FUNCTION_BLOCK FB_Gantry
VAR CONSTANT
	sCycleStateTextDef: ARRAY[0..10]  OF STRING :=	
		['State 0: Wait for Start','1','2','3','4','5','6','7','8','9',
		'State 10: Error'];
	
	tCycleStateTimeouts: ARRAY[0..10] OF TIME := 
		[T#10S,T#10S,T#10S,T#10S,T#10S,T#10S,T#10S,T#10S,T#10S,T#10S,
		T#10S];

	sInitStateTextDef: ARRAY[0..10] OF STRING :=
		['State 0: Wait for Start',
		'State 1: Description Init State 1',
		'State 2: Description Init State 2',
		'State 3; Description Init State 3',
		'State 4; Description Init State 4',
		'State 5; Description Init State 5',
		'State 6; Error State'];

	tInitStateTimeouts: ARRAY[0..10] OF TIME := 
		[T#10S,T#10S,T#10S,T#10S,T#10S,T#10S,T#10S,T#10S,T#10S,T#10S
		,T#10S];
END_VAR
VAR_INPUT
	mxResetCycleState				: BOOL;
	mxResetInitState				: BOOL;
	mxForceInit						: BOOL; (*Reset Calibration Flag*)
	mxReset							: BOOL;	(*Reset Error*)
	mxEmergency						: BOOL;
	mxAutoMode						: BOOL; (* TRUE = Automode *)
	mxFirstCycle					: BOOL;

	mrModPosConveyor				: LREAL;
	mxProductReadyAtTakeout			: BOOL; (* Signal from BottomMold, Takeout Unit *)
	mxDisableCollision				: BOOL;
END_VAR
VAR_IN_OUT
	MachParameters					: ST_GantryMachPar;
	ProdParameters					: ST_GantryProdPar;
	SysParameters					: ST_GantrySysPar;
END_VAR
VAR_OUTPUT
	(*Errors*)
	Errors							: ST_GantryErrors;
	mxErrorInit						: BOOL;		(* Error, stop immediately. Initialisation neccesary *)
	mxErrorStopinPos				: BOOL;		(* Error, stop in position. Only reset neccesary *)

(* State vars *)
	mxCycleBusy						: BOOL;
	mxInitBusy						: BOOL;
	
(* Vars *)
	mxInitialized					: BOOL;
	mrActPosHorizontal				: LREAL;
	mrActPosVertical				: LREAL;
	mxHorizontalIsMoving			: BOOL;
	mxVerticalIsMoving				: BOOL;
	
	(* Signals *)
	mxIsEmpty						: BOOL;
	mxProductPickedUp				: BOOL;
END_VAR
VAR
(* State vars *)
	miCycleState					: INT :=0;
	miCycleOldstate					: INT :=0;
	mxCycleTransitionState			: BOOL := FALSE;
	sCycleStateText					: STRING;
	exCycleTimeOut					: BOOL;		(* Timeout for the whole programcycle *)
	CycleTimeout					: TON;
	CycleTimeOutUpFlank				: R_TRIG;
	mxCycleTimeoutEnable			: BOOL;
	CycleTime						: REAL;
	mxCycleHasError					: BOOL;
	miStopState						: INT;
	mxStartCycle					: BOOL;
	mxStopCycle						: BOOL;
	mxStopDirect					: BOOL;
	
	miInitState						: INT	:=0;
	miInitOldstate					: INT	:=0;
	mxInitTransitionState			: BOOL	:= FALSE;
	sInitStateText					: STRING;
	exInitTimeOut					: BOOL;		(* Timeout for the whole programcycle *)
	InitTimeout						: TON;
	InitTimeOutUpFlank				: R_TRIG;
	mxInitTimeoutEnable				: BOOL;
	InitTime						: REAL;
	mxInitHasError					: BOOL;
	mxStartInit						: BOOL;
	mxStopInit						: BOOL;

	ixCollision						AT %I*: BOOL;	(* Vertical axis *)
	ixEndLimitHorFront				AT %I*: BOOL;
	ixEndLimitHorBack				AT %I*: BOOL;
	ixEndLimitVertUp				AT %I*: BOOL;
	ixEndLimitVertDown				AT %I*: BOOL;
	
	(* Objects *)
	HorizontalAxis					: FB_NcAxis;
	VerticalAxis					: FB_NcAxis;
	(* Pickup Head *)
	BlowOff							: ARRAY [1..6] OF FB_MonoValveNoFdbck;
	VacuumValve						: ARRAY [1..6] OF FB_MonoValveNoFdbck;
	ixVacuumSensor					 AT %I* : ARRAY [1..6] OF BOOL;

(* Vars *)	
	miVacSection					: INT;
	miBlowOffSection				: INT;
	
	mxSwitchVacuumOn				: BOOL;
	(* Errors *)
	SR_exCollision					: SR;
	SR_exEndLimitHorFront			: SR;
	SR_exEndLimitHorBack			: SR;
	SR_exEndLimitVertUp				: SR;
	SR_exEndLimitVertDown			: SR;
	SR_exProductLost				: ARRAY [1..6] OF SR;
	T_VacSensor						: ARRAY [1..6] OF TON;
	mxSwitchBlowOffOn				: BOOL;
	T_WaitAtPickupPosition: TON;
	RT_DropOffPosCoveyor: R_TRIG;
	T_BlowOff: TON;
	mxTemp: BOOL;
	mxTemp2: BOOL;
	mxTest: BOOL;
	FT_SwitchVacuumOff: F_TRIG;
	FT_SwitchBlowOff: F_TRIG;
END_VAR

Error();
Cycle();
Init();
Objects();

ACTION Cycle:
(*StateChange (Transition)  Signalgeneration*)
mxCycleTransitionState:=(miCycleState<>miCycleOldstate);
(*State text*)
sCycleStateText:=sCycleStateTextDef[miCycleState];
(*Timeout Watchdog for Statemachine*)
mxCycleTimeoutEnable:=NOT (miCycleState=0) AND NOT mxReset;

CycleTimeout(IN:=mxCycleTimeoutEnable, PT:=tCycleStateTimeouts[miCycleState] );
CycleTimeOutUpFlank(CLK:=CycleTimeout.Q );
miCycleOldstate:=miCycleState;

(*Set Errorbit when Raising edge of Timeout has been detected*)
IF CycleTimeOutUpFlank.Q THEN
	exCycleTimeOut:=TRUE; 			(* 1 Timeout for the whole programcycle *)
END_IF

(*Function to reset the Statemachine*)
IF mxResetCycleState THEN
	mxResetCycleState:= FALSE;
	miCycleState:=0;
	miCycleOldstate:=miCycleState;
	mxCycleTransitionState:=FALSE;

	mxInitialized:= FALSE;
	mxStartCycle:= FALSE;
	mxStopCycle:= FALSE;
	mxStopDirect:= FALSE;

	mxIsEmpty:= FALSE;
	mxProductPickedUp:= FALSE;
	mxSwitchBlowOffOn:= FALSE;
	mxSwitchVacuumOn:= FALSE;

	T_WaitAtPickupPosition.IN:= FALSE;
	T_BlowOff.IN:= FALSE;
END_IF

fT_SwitchVacuumOff(CLK:= mxSwitchVacuumOn);
FT_SwitchBlowOff(CLK:=mxSwitchBlowOffOn);


(*Definition State has Error*)
mxCycleHasError:=FALSE;

// Open active valves on switch vacuum on.
IF (mxSwitchVacuumOn AND mxAutoMode) THEN
	IF MachParameters.EnableVacuumSection[1] THEN VacuumValve[1].M_On(); END_IF
	IF MachParameters.EnableVacuumSection[2] THEN VacuumValve[2].M_On(); END_IF
	IF MachParameters.EnableVacuumSection[3] THEN VacuumValve[3].M_On(); END_IF
	IF MachParameters.EnableVacuumSection[4] THEN VacuumValve[4].M_On(); END_IF
END_IF

// On trigger, close active valves
IF fT_SwitchVacuumOff.q AND mxAutoMode THEN
	IF MachParameters.EnableVacuumSection[1] THEN VacuumValve[1].M_Off(); END_IF
	IF MachParameters.EnableVacuumSection[2] THEN VacuumValve[2].M_Off(); END_IF
	IF MachParameters.EnableVacuumSection[3] THEN VacuumValve[3].M_Off(); END_IF
	IF MachParameters.EnableVacuumSection[4] THEN VacuumValve[4].M_Off(); END_IF
END_IF

// Open blowoff valves
IF mxSwitchBlowOffOn AND mxAutoMode THEN
	BlowOff[1].M_On();
	BlowOff[2].M_On();
	BlowOff[3].M_On();
	BlowOff[4].M_On();
END_IF

// On trigger, close blowoff valves.
IF FT_SwitchBlowOff.q AND mxAutoMode THEN
	BlowOff[1].M_Off();
	BlowOff[2].M_Off();
	BlowOff[3].M_Off();
	BlowOff[4].M_Off();
END_IF

RT_DropOffPosCoveyor(CLK:= mrModPosConveyor > MachParameters.DropOffConveyorPostion);
T_WaitAtPickupPosition(IN:= , PT:= T#1S);		
T_BlowOff(IN:= , PT:= ProdParameters.BlowOffTime);
IF T_BlowOff.Q THEN T_BlowOff.IN:= FALSE; END_IF
	
(*Cycle State's*)
CASE miCycleState OF
	0:
	(*
	
	- StopCyle en mxPause -> stop bewegingen.
	- Stop Cycle -> empty machine, ga naar rust
	
		- wait for startcycle
		- wait for product ready at takeout
		- Move horizontal to product pickup
		- move vertical to product pickup
		- Vacuum on
		- Move vertical up to transport pos
		- Move horizontal to drop off position (Rest)
		- wait for drop off position conveyor
		- Move vertical down to dropoff position
		- Blow off product
		- Move vertical up to transport pos
		- Goto 1

		* During vertical down, guard the collission sensor=> stop hor and vertical
		* Vacuum sensor check when vacuum on=> error leakage
		*  
	*)
		IF mxStartCycle THEN
			mxStartCycle:= FALSE;
			mxIsEmpty:= FALSE;
			mxProductPickedUp:= FALSE;

			miCycleState:= 1;
		END_IF	

	(* Set when goto 1 mxIsEmpty:= FALSE;	*)

	(* Wait for product ready at takeout *)
	1:
		IF mxStopDirect THEN
			mxStopDirect:= FALSE;
			
			miCycleState:= 25;
		//ELSIF mxStopCycle AND mxPause THEN
		//	mxPause:= FALSE;
			
		//	miCycleState:= 0;
		ELSIF mxStopCycle THEN
			mxStopCycle:= FALSE;
			VerticalAxis.M_Stop();
			HorizontalAxis.M_Stop();
			
			miStopState:= miCycleState;
			miCycleState:= 20;
		ELSIF mxProductReadyAtTakeout THEN
			mxProductReadyAtTakeout:= FALSE;
			mxIsEmpty:= FALSE;
			mxProductPickedUp:= FALSE;
			
			miCycleState:= 2;
		END_IF
		
	(* Move horizontal to the front to pickup position *)
	2:
		IF mxStopDirect THEN
			mxStopDirect:= FALSE;
			
			miCycleState:= 25;
		ELSIF mxStopCycle THEN
			mxStopCycle:= FALSE;
			VerticalAxis.M_Stop();
			HorizontalAxis.M_Stop();
			
			miStopState:= miCycleState;
			miCycleState:= 20;
		ELSIF HorizontalAxis.M_MoveAbsolute(Position:= MachParameters.PositionHorizontalPickup, Velocity:= MachParameters.Hor_VelocityAuto) THEN

			mxSwitchVacuumOn:= TRUE;
			
			miCycleState:=3;
		END_IF

	(* Move Vertical down to pickup position, vacuum on *)
	3:
		IF mxStopDirect THEN
			mxStopDirect:= FALSE;
			
			miCycleState:= 25;
		ELSIF mxStopCycle THEN
			mxStopCycle:= FALSE;
			
			miStopState:= miCycleState;
			miCycleState:= 20;
		ELSIF VerticalAxis.M_MoveAbsolute(Position:= ProdParameters.PositionVerticalPickup, Velocity:= MachParameters.Vert_VelocityAuto) THEN
		
			miCycleState:= 4;
		END_IF

	(* Wait at pickup position *)	
	4:
		T_WaitAtPickupPosition.IN:= TRUE;
	
		IF mxStopDirect THEN
			mxStopDirect:= FALSE;
			
			miCycleState:= 25;
		ELSIF mxStopCycle THEN
			mxStopCycle:= FALSE;
			
			miStopState:= miCycleState;
			miCycleState:= 20;
		ELSIF T_WaitAtPickupPosition.Q THEN
			T_WaitAtPickupPosition.IN:= FALSE;
			
			miCycleState:= 5;
		END_IF		

	(* Move Vertical up to transport position *)
	5:
		IF mxStopDirect THEN
			mxStopDirect:= FALSE;
			
			miCycleState:= 25;
		ELSIF mxStopCycle THEN
			mxStopCycle:= FALSE;
			
			miStopState:= miCycleState;
			miCycleState:= 20;
		ELSIF VerticalAxis.M_MoveAbsolute(Position:= MachParameters.Vert_PositionTransport, Velocity:= MachParameters.Vert_VelocityAuto) THEN
			mxProductPickedUp:= TRUE;

			miCycleState:= 6;
		END_IF
		
	(* Move horizontal to the back to drop-off position *)
	6:
		IF mxStopDirect THEN
			mxStopDirect:= FALSE;
			
			miCycleState:= 25;
		ELSIF mxStopCycle THEN
			mxStopCycle:= FALSE;
			
			miStopState:= miCycleState;
			miCycleState:= 20;
		ELSIF HorizontalAxis.M_MoveAbsolute(Position:= MachParameters.PositionHorizontalDropOff, Velocity:= MachParameters.Hor_VelocityAuto) THEN
			mxProductPickedUp := FALSE;
			miCycleState:= 7;
		END_IF
		
	(* Wait for drop off position conveyor *)
	7:
		IF mxStopDirect THEN
			mxStopDirect:= FALSE;
			
			miCycleState:= 25;
		ELSIF mxStopCycle THEN
			mxStopCycle:= FALSE;
			
			miStopState:= miCycleState;
			miCycleState:= 20;
		ELSIF RT_DropOffPosCoveyor.Q THEN
			
			miCycleState:= 8;
		END_IF

	(* Move Vertical Axis down to drop off position *)
	8:
		IF mxStopDirect THEN
			mxStopDirect:= FALSE;
			
			miCycleState:= 25;
		ELSIF mxStopCycle THEN
			mxStopCycle:= FALSE;
			
			miStopState:= miCycleState;
			miCycleState:= 20;
		ELSIF VerticalAxis.M_MoveAbsolute(Position:= ProdParameters.PositionVerticalDropOff, Velocity:= MachParameters.Vert_VelocityAuto) THEN
			T_BlowOff.IN:= TRUE;
			mxSwitchBlowOffOn := TRUE;
			mxSwitchVacuumOn := FALSE; // bateu 20180619
			
			miCycleState:= 9;
		END_IF
		
	(* Move Vertical Axis up to transport position *)
	9:
		IF mxStopDirect THEN
			mxStopDirect:= FALSE;
			
			miCycleState:= 25;
		ELSIF mxStopCycle THEN
			mxStopCycle:= FALSE;
			
			miStopState:= miCycleState;
			miCycleState:= 20;
		ELSIF T_BlowOff.q THEN
			T_BlowOff.IN := FALSE;
			mxSwitchBlowOffOn := FALSE;
			miCycleState:= 10;
		END_IF
	
	10:
		IF mxStopDirect THEN
			mxStopDirect:= FALSE;
			
			miCycleState:= 25;
		ELSIF mxStopCycle THEN
			mxStopCycle:= FALSE;
			
			miStopState:= miCycleState;
			miCycleState:= 20;
		ELSIF VerticalAxis.M_MoveAbsolute(Position:= MachParameters.Vert_PositionTransport, Velocity:= MachParameters.Vert_VelocityAuto) THEN
			//mxIsEmpty:= TRUE;
			
			miCycleState:= 11;
		END_IF

	(* Move Horizontal Axis to rest position *)
	11:
		IF mxStopDirect THEN
			mxStopDirect:= FALSE;
			
			miCycleState:= 25;
		ELSIF mxStopCycle THEN
			mxStopCycle:= FALSE;
			
			miStopState:= miCycleState;
			miCycleState:= 20;
		ELSIF HorizontalAxis.M_MoveAbsolute(Position:= MachParameters.Hor_Positionrest, Velocity:= MachParameters.Hor_VelocityAuto) THEN
			mxIsEmpty:= TRUE;
			
			miCycleState:= 1;
		END_IF

	(* Stop Cycle *)
	20:
		IF mxStopDirect THEN
			mxStopDirect:= FALSE;
			
			miCycleState:= 21;
		ELSE 
			VerticalAxis.M_Stop();
			HorizontalAxis.M_Stop();
			
			miCycleState:= 21;
		END_IF
	
	(* Stop Cycle, wait for gantry's stopped *)
	21:
		IF mxStopDirect THEN
			mxStopDirect:= FALSE;
			
			miCycleState:= 21;
		ELSIF (HorizontalAxis.axStatus.StandStill OR NOT HorizontalAxis.axStatus.Moving) AND (VerticalAxis.axStatus.StandStill OR NOT VerticalAxis.axStatus.Moving) THEN
			
			miCycleState:= 22;
		END_IF

	(* Stop Cycle, wait for restart *)
	22:
		IF mxStopDirect THEN
			mxStopDirect:= FALSE;
			
			miCycleState:= 21;
		ELSIF mxStartCycle THEN
			mxStartCycle:= FALSE;
			
			miCycleState:= miStopState;
		END_IF

	(* Stop Direct *)
	25:
		mxInitialized:= FALSE;
		mxStartCycle:= FALSE;
		mxStopCycle:= FALSE;
		mxStopDirect:= FALSE;

		mxIsEmpty:= FALSE;
		mxProductPickedUp:= FALSE;
		mxSwitchBlowOffOn:= FALSE;
		mxSwitchVacuumOn:= FALSE;

		T_WaitAtPickupPosition.IN:= FALSE;
		T_BlowOff.IN:= FALSE;

		miCycleState:= 0;
END_CASE

mxCycleBusy:= miCycleState<>0 AND NOT (miCycleState=22);
END_ACTION

ACTION Error:
SR_exCollision(SET1:= NOT ixCollision AND NOT mxDisableCollision, RESET:= mxReset, Q1=> Errors.Collision);
SR_exEndLimitHorFront(SET1:= NOT ixEndLimitHorFront, RESET:= mxReset, Q1=> Errors.EndLimitHorFront);
SR_exEndLimitHorBack(SET1:= NOT ixEndLimitHorBack, RESET:= mxReset, Q1=> Errors.EndLimitHorBack);
SR_exEndLimitVertUp(SET1:= NOT ixEndLimitVertUp, RESET:= mxReset, Q1=> Errors.EndLimitVertUp);
SR_exEndLimitVertDown(SET1:= NOT ixEndLimitVertDown, RESET:= mxReset, Q1=> Errors.EndLimitVertDown);

(*
FOR miVacSection:= 1 TO 6 DO
T_VacSensor[miVacSection](IN:= VacuumValve[miVacSection].mxIsOn, PT:= T#3S);
SR_exProductLost[miVacSection](
		SET1:= MachParameters.EnableVacuumSection[miVacSection] AND VacuumValve[miVacSection].mxIsOn AND (T_VacSensor[miVacSection].Q AND NOT ixVacuumSensor[miVacSection]) , 
		RESET:= mxReset, Q1=> Errors.ProductLost[miVacSection]);
END_FOR
*)

T_VacSensor[1](IN:= VacuumValve[1].mxIsOn, PT:= T#3S);
SR_exProductLost[1](
		SET1:= MachParameters.EnableVacuumSection[1] AND VacuumValve[1].mxIsOn AND (T_VacSensor[1].Q AND NOT ixVacuumSensor[1]) , 
		RESET:= mxReset, Q1=> Errors.ProductLost[1]);
		
T_VacSensor[2](IN:= VacuumValve[2].mxIsOn, PT:= T#3S);
SR_exProductLost[2](
		SET1:= MachParameters.EnableVacuumSection[2] AND VacuumValve[2].mxIsOn AND (T_VacSensor[2].Q AND NOT ixVacuumSensor[2]) , 
		RESET:= mxReset, Q1=> Errors.ProductLost[2]);
		
T_VacSensor[3](IN:= VacuumValve[3].mxIsOn, PT:= T#3S);
SR_exProductLost[3](
		SET1:= MachParameters.EnableVacuumSection[3] AND VacuumValve[3].mxIsOn AND (T_VacSensor[3].Q AND NOT ixVacuumSensor[3]) , 
		RESET:= mxReset, Q1=> Errors.ProductLost[3]);
		
T_VacSensor[4](IN:= VacuumValve[4].mxIsOn, PT:= T#3S);
SR_exProductLost[4](
		SET1:= MachParameters.EnableVacuumSection[4] AND VacuumValve[4].mxIsOn AND (T_VacSensor[4].Q AND NOT ixVacuumSensor[4]) , 
		RESET:= mxReset, Q1=> Errors.ProductLost[4]);






(*************************************************************************************************)
mxErrorInit:= Errors.Collision OR Errors.EndLimitHorFront OR Errors.EndLimitHorBack OR Errors.EndLimitVertUp OR Errors.EndLimitVertDown OR
	HorizontalAxis.ErrorStop OR VerticalAxis.ErrorStop;;
mxErrorStopinPos:= FALSE;
END_ACTION

ACTION Init:
(*StateChange (Transition)  Signalgeneration*)
mxInitTransitionState:=(miInitState<>miInitOldstate);
(*State text*)
sInitStateText:=sInitStateTextDef[miInitState];
(*Timeout Watchdog for Statemachine*)
mxInitTimeoutEnable:=NOT (miInitState=0)  AND NOT mxReset;

InitTimeout(IN:=mxInitTimeoutEnable  , PT:=tInitStateTimeouts[miInitState] );
InitTimeOutUpFlank(CLK:=InitTimeout.Q );
miInitOldstate:=miInitState;

(*Set Errorbit when Raising edge of Timeout has been detected*)
IF InitTimeOutUpFlank.Q THEN
	exInitTimeOut:=TRUE; 			(* 1 Timeout for the whole programcycle *)
END_IF

(*Function to reset the Statemachine*)
IF mxResetInitState THEN
	mxResetInitState:=FALSE;
	miInitState:=0;
	miInitOldstate:=miInitState;
	mxInitTransitionState:=FALSE;

	mxInitialized:= FALSE;	
	mxStartInit:= FALSE;
	mxStopInit:= FALSE;
END_IF

(*Definition State has Error*)
mxInitHasError:=FALSE;

(*Init State's*)
CASE miInitState OF
	0:
	
	(* 
		- Wait for start int
		- Blow off uit
		- vacuum aan laten
		- Vertical move up to transport pos.
		- Horizontal move back to drop off positie
		- 	
	
	*)
		IF mxStartInit THEN
			mxStartInit:= FALSE;
			mxInitialized:= FALSE;

			(* Don't turn vacuum off, turn blowoff off *)
			mxSwitchBlowOffOn:= FALSE;
			
			miInitState:= 1;
		END_IF

	(* Move vertical up *)
	1:
		IF mxStopInit THEN
			mxStopInit:= FALSE;
			
			miInitState:= 10;
		ELSIF VerticalAxis.M_MoveAbsolute(Position:= MachParameters.Vert_PositionTransport, Velocity:= MachParameters.Vert_VelocityAuto) THEN
			
			miInitState:= 2;			
		END_IF

	(* Move horizontal back *)
	2:
		IF mxStopInit THEN
			mxStopInit:= FALSE;

			miInitState:= 10;
		ELSIF HorizontalAxis.M_MoveAbsolute(Position:= MachParameters.Hor_Positionrest, Velocity:= MachParameters.Hor_VelocityAuto) THEN
			
			mxInitialized:= TRUE;
			miInitState:= 0;			
		END_IF

	(* Stop Init *)
	10:
		mxInitialized:= FALSE;	
		mxStartInit:= FALSE;
		mxStopInit:= FALSE;

		VerticalAxis.M_Stop();
		HorizontalAxis.M_Stop();
		
		miInitState:= 0;
		
END_CASE

mxInitBusy:= miInitState<>0;
END_ACTION

METHOD M_StartCycle

IF NOT mxCycleBusy THEN
	mxStartCycle:= TRUE;	
END_IF
END_METHOD

METHOD M_StartInit
VAR_INPUT
END_VAR

IF NOT mxInitBusy THEN
	mxStartInit:= TRUE;
END_IF
END_METHOD

METHOD M_StopCycle

IF mxCycleBusy THEN 
	mxStopCycle:= TRUE; 
END_IF
END_METHOD

METHOD M_StopDirect

IF mxCycleBusy THEN
	mxStopDirect:= TRUE;	
END_IF
END_METHOD

METHOD M_StopInit

IF mxInitBusy THEN 
	mxStopInit:= TRUE; 
END_IF
END_METHOD

ACTION Objects:
HorizontalAxis(
	mxEnable:= NOT mxEmergency, 
	mxInhibit:= FALSE, 
	mxAutoMode:= mxAutoMode, 
	mxReset:= mxReset, 
	mxFirstCycle:= 	mxFirstCycle,
	mxEmergency:= mxEmergency, 
	mxSimulation:= , 
	mxResetCycle:= , 
	mxDisable_Positive:= NOT ixEndLimitHorFront, 
	mxDisable_Negative:= NOT ixEndLimitHorBack, 
	mxBlockHMI:= , 
	mrOverride:= 100.0,
	mrVelocityManual:= MachParameters.Hor_VelocityManual,
	mrHomePos:= MachParameters.Hor_PositionHome, 
	SysParameters:= SysParameters.HorizontalAxis,
	mxCycleBusy=> , 
	mxRunning=> , 
	Errors=> Errors.HorizontalNCAxisError, 
	Error=> , 
	ErrorStop=> , 
	axStatus=> , 
	mxAxisIsMoving=> mxHorizontalIsMoving,
	ActPosition=> mrActPosHorizontal, 
	ActVelocity=> , 
	axAxis=> );
	
VerticalAxis(
	mxEnable:= NOT mxEmergency, 
	mxInhibit:= FALSE, 
	mxAutoMode:= mxAutoMode, 
	mxReset:= mxReset, 
	mxFirstCycle:= 	mxFirstCycle,
	mxEmergency:= mxEmergency, 
	mxSimulation:= , 
	mxResetCycle:= , 
	mxDisable_Positive:= NOT ixEndLimitVertUp, 
	mxDisable_Negative:= (NOT ixEndLimitVertDown) OR Errors.Collision, 
	mxBlockHMI:= , 
	mrOverride:= 100.0, 
	mrVelocityManual:= MachParameters.Vert_VelocityManual, 
	mrHomePos:= MachParameters.Vert_PositionHome, 
	SysParameters:= SysParameters.VerticalAxis,
	mxCycleBusy=> , 
	mxRunning=> , 
	Errors=> Errors.VerticalNCAxisError, 
	Error=> , 
	ErrorStop=> , 
	axStatus=> , 
	mxAxisIsMoving=> mxVerticalIsMoving,
	ActPosition=> mrActPosVertical, 
	ActVelocity=> , 
	axAxis=> );

FOR miVacSection:= 1 TO 6 DO	
	VacuumValve[miVacSection](
		mxReset:= mxReset, 
		mxEmergency:= mxEmergency, 
		mxAutoMode:= mxAutoMode, 
		mxIsOn=> );
END_FOR
FOR miBlowOffSection:= 1 TO 6 DO
	BlowOff[miBlowOffSection](
		mxReset:= mxReset, 
		mxEmergency:= mxEmergency, 
		mxAutoMode:= mxAutoMode, 
		mxIsOn=> );
END_FOR
END_ACTION

END_FUNCTION_BLOCK

(* stored: Version 1.1.0.1, ProductVersion 3.1.4020.12
   POU FB_Gantry: Id {ec7f78dd-5062-47e3-8cb6-2a2e0ceb8133}, SpecialFunc None
   Action Cycle: Id {40de9b08-53c7-4a15-bbb0-3796579dcb28}
   Action Error: Id {05bb1052-d95e-4ab8-8ba0-ccbc2e4ec32c}
   Action Init: Id {881751bc-85ad-412a-b591-7b792cb81755}
   Method M_StartCycle: Id {b3d619fb-9a6a-470c-af33-50adf215b18b}
   Method M_StartInit: Id {7bd8aafa-511b-4a28-b95d-080cb2f9f6bf}
   Method M_StopCycle: Id {7d44c36c-e6eb-473d-ba72-acaf2ed26a6b}
   Method M_StopDirect: Id {a9f40ebc-f527-4cd7-86f5-d61f2c026935}
   Method M_StopInit: Id {c07af727-e87e-4ef4-8512-cc5f9ac6ac46}
   Action Objects: Id {b346841c-6e61-425f-9976-22029e62eb23} *)
